PROGRAM MAIN
VAR
	values : ARRAY [0..24] OF LREAL;
	i : INT;
END_VAR

values[0] := values[0] + 1;

IF values[0] > 100 THEN
	values[0] := 0;
END_IF

FOR i := 1 TO 24 DO
	values[i] := values[0] + (i * 10);
	
	gvl.arrayWithStructureWithArray[0].myArray[0] := values[0];
	gvl.structureWithArray.myArray[0] := values[0];
	gvl.structureWithStructureWithArray.myStruct.myArray[0] := values[0];
	
END_FOR

END_PROGRAM

(* stored: Version 1.1.0.1, ProductVersion 3.1.4024.11
   POU MAIN: Id {d4424a59-9d68-4c5d-8978-6f205cb721c5}, SpecialFunc None *)
